PROGRAM P_Inputs
VAR
	fbJoystickWinch 				: FB_JoystickInputScaling;
	fbJoystickCyl 					: FB_JoystickInputScaling;
	fbJoystickRot 					: FB_JoystickInputScaling;
	fbWinchPosition 				: FB_Encoder;
	fbCylinderPosition 				: FB_Encoder;
	fbCylPistonPosition 			: FB_AnalogInputScaling;
	fbPressureSupply 				: FB_AnalogInputScaling;
	fbPressureReturn 				: FB_AnalogInputScaling;
	fbPressureCyl_A_PistonSide 		: FB_AnalogInputScaling;
	fbPressureCyl_B_RodSide			: FB_AnalogInputScaling;
	fbPressureWinch_A1_Input 		: FB_AnalogInputScaling;
	fbPressureWinch_A2_Input 		: FB_AnalogInputScaling;
	fbPressureWinch_B_Output		: FB_AnalogInputScaling;
	eStatus : E_Status;
END_VAR

fbJoystickWinch(
	bEnable := G_IO.bManualSwtich,
	nRawInput := G_IO.fJoyYraw,
	stJoystickInputScaling := G_Parameters.stParam.stJoystickInputScalingY,
	fNormalizedOutput => G_Sensors.fJoystickNormalizedY
);

fbJoystickCyl(
	bEnable := G_IO.bManualSwtich,
	nRawInput := G_IO.fJoyXraw,
	stJoystickInputScaling := G_Parameters.stParam.stJoystickInputScalingX,
	fNormalizedOutput => G_Sensors.fJoystickNormalizedX
);

fbJoystickRot(
	bEnable := G_IO.bManualSwtich,
	nRawInput := G_IO.fJoyZraw,
	stJoystickInputScaling := G_Parameters.stParam.stJoystickInputScalingZ,
	fNormalizedOutput => G_Sensors.fJoystickNormalizedZ
);

fbWinchPosition (
	nRawInput := G_IO.nWinchEncoderValue, 
	fEncoderOffset := G_Parameters.stParam.fWinchEncoderOffset,
	fPosition => G_Sensors.fWinchEncoderPosition
);

fbCylinderPosition (
	nRawInput := G_IO.nCylinderEncoderValue, 
	fEncoderOffset := G_Parameters.stParam.fCylinderEncoderOffset,
	fPosition => G_Sensors.fCylinderEncoderPosition
);

//G_Sensors.fWinchWirePosition := fbWinchPosition.fPosition*G_Parameters.stParam.fWinchDrumScaling;
G_Sensors.fCylinderPosition := -(fbCylinderPosition.fPosition/360)*G_Parameters.stParam.fCylinderDrawWireGearRadius*0.001;


fbPressureSupply(
	nRawInput := G_IO.fPressureSupply,
	stAnalogInputScaling := G_Parameters.stParam.stPressureSensorScaling400bar,
	fOutput => G_Sensors.fPressureSupply
);

fbPressureReturn(
	nRawInput := G_IO.fPressureReturn,
	stAnalogInputScaling := G_Parameters.stParam.stPressureSensorScaling40bar,
	fOutput => G_Sensors.fPressureReturn
);

fbPressureCyl_A_PistonSide(
	nRawInput := G_IO.fPressureCylinderA,
	stAnalogInputScaling := G_Parameters.stParam.stPressureSensorScaling400bar,
	fOutput => G_Sensors.fPressureCylinderA
);

fbPressureCyl_B_RodSide(
	nRawInput := G_IO.fPressureCylinderB,
	stAnalogInputScaling := G_Parameters.stParam.stPressureSensorScaling400bar,
	fOutput => G_Sensors.fPressureCylinderB
);

fbPressureWinch_A1_Input(
	nRawInput := G_IO.fPressureWinchA1,
	stAnalogInputScaling := G_Parameters.stParam.stPressureSensorScaling400bar,
	fOutput => G_Sensors.fPressureWinchA1
);

fbPressureWinch_A2_Input(
	nRawInput := G_IO.fPressureWinchA2,
	stAnalogInputScaling := G_Parameters.stParam.stPressureSensorScaling400bar,
	fOutput => G_Sensors.fPressureWinchA2
);

fbPressureWinch_B_Output(
	nRawInput := G_IO.fPressureWinchB,
	stAnalogInputScaling := G_Parameters.stParam.stPressureSensorScaling400bar,
	fOutput => G_Sensors.fPressureWinchB
);

END_PROGRAM

(* stored: Version 1.1.0.1, ProductVersion 3.1.4024.12
   POU P_Inputs: Id {8b676dbd-393f-42d6-8803-330b6e90ab14}, SpecialFunc None *)
